# EPICS substitutions: gigeApp/Db/autosave_gige.substitutions
#
# gige substitutions file
#

# Generate iocAdmin autosave request
file autosave_iocAdmin.template
{
    {
        IOC     =   $(IOC)
    }
}

# Generate one set per camera
file autosave_gige.template
{
    {   CAM     =   13PS1  }
}
